ABB RAPID module: 003D1A03

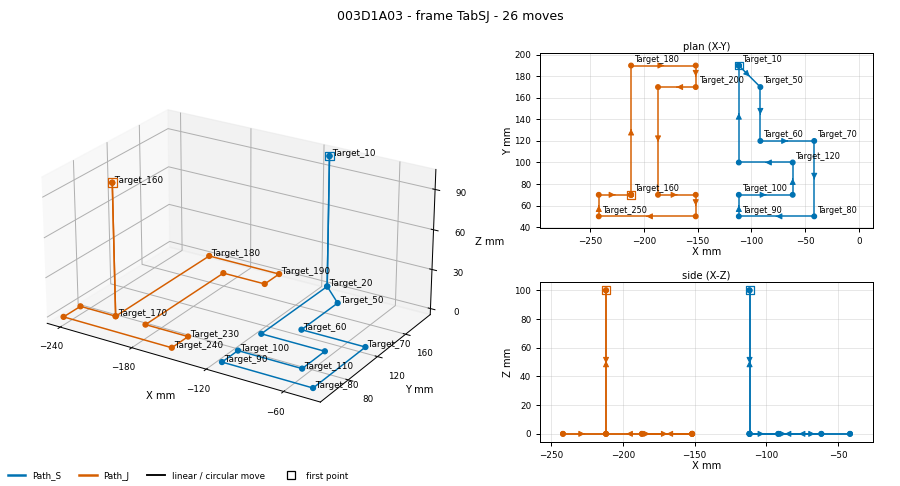
[picture p0: tool path of 003D1A03 in frame TabSJ, 26 of 28 moves have a stored position in this frame; points joined in program order, loops and branches not executed]
MODULE Module1
	CONST robtarget Target_10:=[[-111.75,190.000000035,99.999999935],[0,0.707106781,0.707106781,0],[0,0,0,0],[9E+09,9E+09,9E+09,9E+09,9E+09,9E+09]];
	CONST robtarget Target_20:=[[-111.75,190,-0.000000065],[0,0.707106781,0.707106781,0],[0,0,0,0],[9E+09,9E+09,9E+09,9E+09,9E+09,9E+09]];
	CONST robtarget Target_30:=[[-41.75,190,-0.000000065],[0,0.707106781,0.707106781,0],[0,0,0,0],[9E+09,9E+09,9E+09,9E+09,9E+09,9E+09]];
	CONST robtarget Target_40:=[[-41.75,170,-0.000000057],[0,0.707106781,0.707106781,0],[0,0,0,0],[9E+09,9E+09,9E+09,9E+09,9E+09,9E+09]];
	CONST robtarget Target_50:=[[-91.75,170,-0.000000057],[0,0.707106781,0.707106781,0],[0,0,0,0],[9E+09,9E+09,9E+09,9E+09,9E+09,9E+09]];
	CONST robtarget Target_60:=[[-91.75,120,-0.000000041],[0,0.707106781,0.707106781,0],[0,0,0,0],[9E+09,9E+09,9E+09,9E+09,9E+09,9E+09]];
	CONST robtarget Target_70:=[[-41.75,120,-0.000000041],[0,0.707106781,0.707106781,0],[0,0,0,0],[9E+09,9E+09,9E+09,9E+09,9E+09,9E+09]];
	CONST robtarget Target_80:=[[-41.75,50,-0.000000017],[0,0.707106781,0.707106781,0],[0,0,0,0],[9E+09,9E+09,9E+09,9E+09,9E+09,9E+09]];
	CONST robtarget Target_90:=[[-111.75,50,-0.000000017],[0,0.707106781,0.707106781,0],[0,0,0,0],[9E+09,9E+09,9E+09,9E+09,9E+09,9E+09]];
	CONST robtarget Target_100:=[[-111.75,70,-0.000000024],[0,0.707106781,0.707106781,0],[0,0,0,0],[9E+09,9E+09,9E+09,9E+09,9E+09,9E+09]];
	CONST robtarget Target_110:=[[-61.75,70,-0.000000024],[0,0.707106781,0.707106781,0],[0,0,0,0],[9E+09,9E+09,9E+09,9E+09,9E+09,9E+09]];
	CONST robtarget Target_120:=[[-61.75,100,-0.000000034],[0,0.707106781,0.707106781,0],[0,0,0,0],[9E+09,9E+09,9E+09,9E+09,9E+09,9E+09]];
	CONST robtarget Target_130:=[[-111.75,100,-0.000000034],[0,0.707106781,0.707106781,0],[0,0,0,0],[9E+09,9E+09,9E+09,9E+09,9E+09,9E+09]];
	CONST robtarget Target_140:=[[-111.75,190,-0.000000065],[0,0.707106781,0.707106781,0],[0,0,0,0],[9E+09,9E+09,9E+09,9E+09,9E+09,9E+09]];
	CONST robtarget Target_150:=[[-111.75,190.000000035,99.999999935],[0,0.707106781,0.707106781,0],[0,0,0,0],[9E+09,9E+09,9E+09,9E+09,9E+09,9E+09]];
	CONST robtarget Target_160:=[[-211.75,70.000000034,99.999999976],[0,0.707106781,0.707106781,0],[0,0,0,0],[9E+09,9E+09,9E+09,9E+09,9E+09,9E+09]];
	CONST robtarget Target_170:=[[-211.75,70,-0.000000024],[0,0.707106781,0.707106781,0],[0,0,0,0],[9E+09,9E+09,9E+09,9E+09,9E+09,9E+09]];
	CONST robtarget Target_180:=[[-211.75,190,-0.000000065],[0,0.707106781,0.707106781,0],[0,0,0,0],[9E+09,9E+09,9E+09,9E+09,9E+09,9E+09]];
	CONST robtarget Target_190:=[[-151.75,190,-0.000000065],[0,0.707106781,0.707106781,0],[0,0,0,0],[9E+09,9E+09,9E+09,9E+09,9E+09,9E+09]];
	CONST robtarget Target_200:=[[-151.75,170,-0.000000057],[0,0.707106781,0.707106781,0],[0,0,0,0],[9E+09,9E+09,9E+09,9E+09,9E+09,9E+09]];
	CONST robtarget Target_210:=[[-186.75,170,-0.000000057],[0,0.707106781,0.707106781,0],[0,0,0,0],[9E+09,9E+09,9E+09,9E+09,9E+09,9E+09]];
	CONST robtarget Target_220:=[[-186.75,70,-0.000000024],[0,0.707106781,0.707106781,0],[0,0,0,0],[9E+09,9E+09,9E+09,9E+09,9E+09,9E+09]];
	CONST robtarget Target_230:=[[-151.75,70,-0.000000024],[0,0.707106781,0.707106781,0],[0,0,0,0],[9E+09,9E+09,9E+09,9E+09,9E+09,9E+09]];
	CONST robtarget Target_240:=[[-151.75,50,-0.000000017],[0,0.707106781,0.707106781,0],[0,0,0,0],[9E+09,9E+09,9E+09,9E+09,9E+09,9E+09]];
	CONST robtarget Target_250:=[[-241.75,50,-0.000000017],[0,0.707106781,0.707106781,0],[0,0,0,0],[9E+09,9E+09,9E+09,9E+09,9E+09,9E+09]];
	CONST robtarget Target_260:=[[-241.75,70,-0.000000024],[0,0.707106781,0.707106781,0],[0,0,0,0],[9E+09,9E+09,9E+09,9E+09,9E+09,9E+09]];
	CONST robtarget Target_270:=[[-211.75,70,-0.000000024],[0,0.707106781,0.707106781,0],[0,0,0,0],[9E+09,9E+09,9E+09,9E+09,9E+09,9E+09]];
	CONST robtarget Target_280:=[[-211.75,70.000000034,99.999999976],[0,0.707106781,0.707106781,0],[0,0,0,0],[9E+09,9E+09,9E+09,9E+09,9E+09,9E+09]];
	CONST jointtarget Home:=[[0,0,0,0,0,0],[9E+09,9E+09,9E+09,9E+09,9E+09,9E+09]];
	CONST jointtarget Mid:=[[0,30,0,0,30,0],[9E+09,9E+09,9E+09,9E+09,9E+09,9E+09]];
    !***********************************************************
    !
    ! Módulo:  Module1
    !
    ! Descripción:
    !   <Introduzca la descripción aquí>
    !
    ! Autor: Usuario
    !
    ! Versión: 1.0
    !
    !***********************************************************


    !***********************************************************
    !
    ! Procedimiento Main
    !
    !   Este es el punto de entrada de su programa
    !
    !***********************************************************
    PROC main()
        Path_H;
        Path_M;
        Path_J;
        Path_S;
        Path_M;
        Path_H;
    ENDPROC
	PROC Path_S()
	    MoveL Target_10,v200,z10,TOOLSJTCP\WObj:=TabSJ;
	    MoveL Target_20,v200,z10,TOOLSJTCP\WObj:=TabSJ;
	    !MoveL Target_30,v200,z10,TOOLSJTCP\WObj:=TabSJ;
	    !MoveL Target_40,v200,z10,TOOLSJTCP\WObj:=TabSJ;
	    MoveL Target_50,v200,z10,TOOLSJTCP\WObj:=TabSJ;
	    MoveL Target_60,v200,z10,TOOLSJTCP\WObj:=TabSJ;
	    MoveL Target_70,v200,z10,TOOLSJTCP\WObj:=TabSJ;
	    MoveL Target_80,v200,z10,TOOLSJTCP\WObj:=TabSJ;
	    MoveL Target_90,v200,z10,TOOLSJTCP\WObj:=TabSJ;
	    MoveL Target_100,v200,z10,TOOLSJTCP\WObj:=TabSJ;
	    MoveL Target_110,v200,z10,TOOLSJTCP\WObj:=TabSJ;
	    MoveL Target_120,v200,z10,TOOLSJTCP\WObj:=TabSJ;
	    MoveL Target_130,v200,z10,TOOLSJTCP\WObj:=TabSJ;
	    MoveL Target_140,v200,z10,TOOLSJTCP\WObj:=TabSJ;
	    MoveL Target_150,v200,z10,TOOLSJTCP\WObj:=TabSJ;
	ENDPROC
	PROC Path_J()
	    MoveL Target_160,v200,z10,TOOLSJTCP\WObj:=TabSJ;
	    MoveL Target_170,v200,z10,TOOLSJTCP\WObj:=TabSJ;
	    MoveL Target_180,v200,z10,TOOLSJTCP\WObj:=TabSJ;
	    MoveL Target_190,v200,z10,TOOLSJTCP\WObj:=TabSJ;
	    MoveL Target_200,v200,z10,TOOLSJTCP\WObj:=TabSJ;
	    MoveL Target_210,v200,z10,TOOLSJTCP\WObj:=TabSJ;
	    MoveL Target_220,v200,z10,TOOLSJTCP\WObj:=TabSJ;
	    MoveL Target_230,v200,z10,TOOLSJTCP\WObj:=TabSJ;
	    MoveL Target_240,v200,z10,TOOLSJTCP\WObj:=TabSJ;
	    MoveL Target_250,v200,z10,TOOLSJTCP\WObj:=TabSJ;
	    MoveL Target_260,v200,z10,TOOLSJTCP\WObj:=TabSJ;
	    MoveL Target_270,v200,z10,TOOLSJTCP\WObj:=TabSJ;
	    MoveL Target_280,v200,z10,TOOLSJTCP\WObj:=TabSJ;
	ENDPROC
	PROC Path_H()
	    MoveAbsJ Home,v400,z100,tool0\WObj:=TabSJ;
	ENDPROC
	PROC Path_M()
	    MoveAbsJ Mid,v400,z100,tool0\WObj:=TabSJ;
	ENDPROC
ENDMODULE
